{attribute 'qualified_only'}
{attribute 'strict'}
{attribute 'to_string'}
TYPE ST175_Cylinders_e : 
(
	Niederhalter,
	Door_entry,
	Door_exit,
	_max
);
END_TYPE

(* stored: Version 1.1.0.1, ProductVersion 3.1.4024.6
   EnumerationTextList ST175_Cylinders_e: Id {aeb3b67f-61ea-488b-8dbe-4bc1d16749d7} *)
